// TwinCAT 3 PLC project AdsSyncPlcDemo
// ProgramVersion: 3.1.4024.0
// libraries:
//   Tc2_Standard, * (Beckhoff Automation GmbH)
//   Tc2_System, * (Beckhoff Automation GmbH)
//   Tc3_Module, * (Beckhoff Automation GmbH)
// project tree:
//   DUTs/ _DATA_FROM_HMI.TcDUT (not stored), _DATA_TO_HMI.TcDUT (not stored)
//   GVLs/ GVL.TcGVL (not stored)
//   / PlcTask.TcTTO (not stored)
//   POUs/ MAIN.TcPOU

// ---- POUs/MAIN.TcPOU
PROGRAM MAIN
VAR
	
END_VAR

GVL.DataToHmi.LifeBit			:= GVL.DataFromHmi.LifeBit;
GVL.DataToHmi.TestArray			:= GVL.DataFromHmi.TestArray;
GVL.DataToHmi.TestDouble		:= GVL.DataFromHmi.TestDouble;
GVL.DataToHmi.TestString		:= GVL.DataFromHmi.TestString;

END_PROGRAM
